// TIA Portal V16 export
// export: Created 2024-09-05T17:39:25.164551Z, ExportSetting WithDefaults, DisplayName Totally Integrated Automation Portal, DisplayVersion V16 Update 6, DisplayName TIA Portal Version Control Interface, DisplayVersion V16 Update 2, DisplayName TIA Portal Openness, DisplayVersion V16 Update 6, DisplayName STEP 7 Professional, DisplayVersion V16 Update 6, DisplayName STEP 7 Safety, DisplayVersion V16, DisplayName WinCC Advanced, DisplayVersion V16 Update 6
DATA_BLOCK "MII_Parameters"   // DB2020
{ S7_Optimized_Access := 'TRUE' }
AUTHOR : bartz
VERSION : 0.1
// stored: AutoNumber false, DBAccessibleFromOPCUA true, IsOnlyStoredInLoadMemory false, IsRetainMemResEnabled false, IsWriteProtectedInAS false, MemoryReserve 100
   VAR RETAIN
      Connection : Struct
         IPAddress : WString := WSTRING#'10.223.41.34';   // Server IP Address (e.g. 10.223.41.34)
         ServerPort : WString := WSTRING#'58710/PCoUaServer';   // Server port (e.g. 58710/PCoUaServer) / Server port (e.g. 58710)
         PlantID : WString := WSTRING#'P2';   // Unique plant id defined by local DMC key user (e.g. P1, P2) / Unique plant id defined by local DMC key user (e.g. P1 or P2)
         PLC_ID : WString := WSTRING#'1300T1';   // Unique plc id defined by local DMC key user (different from ijcore)
         OperationMode : Bool;   // False: production; True: test
      END_STRUCT;
   END_VAR
   VAR
      Commands : Struct
         getLocalTime : Bool;   // Forces the call for local time
         testProdDeclaration : Bool;   // Forces the call for production declaration
         auxTestProdDeclaration : Int := 1;   // Auxiliar counter for testing
         forceReconnection : Bool;   // Forces the reconnection to the server
      END_STRUCT;
   END_VAR
   VAR RETAIN
      Connection_Status : Struct
         opcUaConnected : Bool;   // True if the client is connected to the server; False if downgraded mode active / True if the client if connected to the server
         opcUaError : Bool;   // True if error during connection attempt
         opcUaStatus : Word;
         opcUaDiagnostics : DWord;   // Detailled error information / Detailed error information
         aux : Struct
            diagnosticStatus : DInt;   // Diagnostic status
            opcUaSubfunctionStatus : DInt;   // Subfunction status
            nAttemptsTotal : Int := 1;   // Number of reconnection attempts
         END_STRUCT;
      END_STRUCT;
   END_VAR
   VAR
      Variability : Struct
         Inputs : Struct
            equipmentVariability : WString[1];
            businessCode : WString[1];
            technoCode : WString[2];
            stationNumber : WString[1];
            varType : WString[1];
            x : Bool;
         END_STRUCT;
         Output : Struct
            variabilityCode : WString[8];
         END_STRUCT;
      END_STRUCT;
   END_VAR
   VAR RETAIN
      M000_Status : Struct
         error : Bool;   // True if an error has occurred during method call / True if an error occurred during method call
         status : WString;   // Detailled error information / Detailed error information
         timestamp : LDT;   // Timestamp of method call attempt
         Inputs : "MII_Interface.MII_METHODS.M000_PRODUCTION_DECLARATION.Inputs";   // Input arguments during error
         Outputs { S7_SetPoint := 'True'} : "MII_Interface.MII_METHODS.M000_PRODUCTION_DECLARATION.Outputs";   // Output arguments during error
      END_STRUCT;
      M002_Status : Struct
         localTime : LDT;   // Last local time received / Last system time received
         status : WString;   // Status of method call
      END_STRUCT;
   END_VAR
BEGIN
END_DATA_BLOCK
